{attribute 'qualified_only'}
{attribute 'strict'}
TYPE eState_INTER :
(
	init,
    setPositions,
    checkSetPositions,
    goToNeutral,
    CheckNeutral,
    enableSPG,
    checkEnableSPG,
    disableSPG,
    checkDisableSPG,
    operation,
    startRecovery,
    recoveryDefaultPosition,
    waitForRecovery,
    error
);
END_TYPE

(* stored: Version 1.1.0.1, ProductVersion 3.1.4024.11
   DUT eState_INTER: Id {5c829116-f8b2-4b9d-94cf-bbbb41200982} *)
